FUNCTION min_array : LREAL
VAR_IN_OUT
	aData : ARRAY[*] OF LREAL;
END_VAR
VAR
	nIdx: DINT;
END_VAR

min_array := 1.7976931348623158E+308;
FOR nIdx := LOWER_BOUND(aData,1) TO UPPER_BOUND(aData,1) DO
	min_array := MIN(aData[nIdx],min_array);
END_FOR

END_FUNCTION

(* stored: Version 1.1.0.1, ProductVersion 3.1.4024.12
   POU min_array: Id {18d92879-ad6c-4aa9-bffe-8a1a8e3732b8}, SpecialFunc None *)
